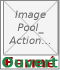
VISUALIZATION Sink  // 60x70
VAR_IN_OUT
	Etat_MaAr	:BOOL;
END_VAR
    Image (3,0 55x55), invisible if: NOT Etat_MaAr, image: ImagePool_Action.Sink_Open
    Image (3,0 55x55), invisible if: Etat_MaAr, image: ImagePool_Action.Sink_Close
    Rectangle (0,55 60x15), "Fermé", invisible if: Etat_MaAr, text list: 'OuvFerm', text index: S_Cmd_ElectroValve_Alim_Lavabo
    Rectangle (0,55 60x15), "Ouvert", invisible if: NOT Etat_MaAr, text list: 'OuvFerm', text index: S_Cmd_ElectroValve_Alim_Lavabo
END_VISUALIZATION

(* stored: Version 1.1.0.1, ProductVersion 3.1.4024.15
   Visu Sink: Id {ba4c94e5-f0e3-4fa6-9c80-6e2b23695f30} *)
